// Mitsubishi GX Works2 project: FB_practice   PLC: Q02/Q02H

PROGRAM MAIN
VAR
  DOUBLE_SOL_1 : DOUBLE_SOL;
  DOUBLE_SOL_2 : DOUBLE_SOL;
END_VAR
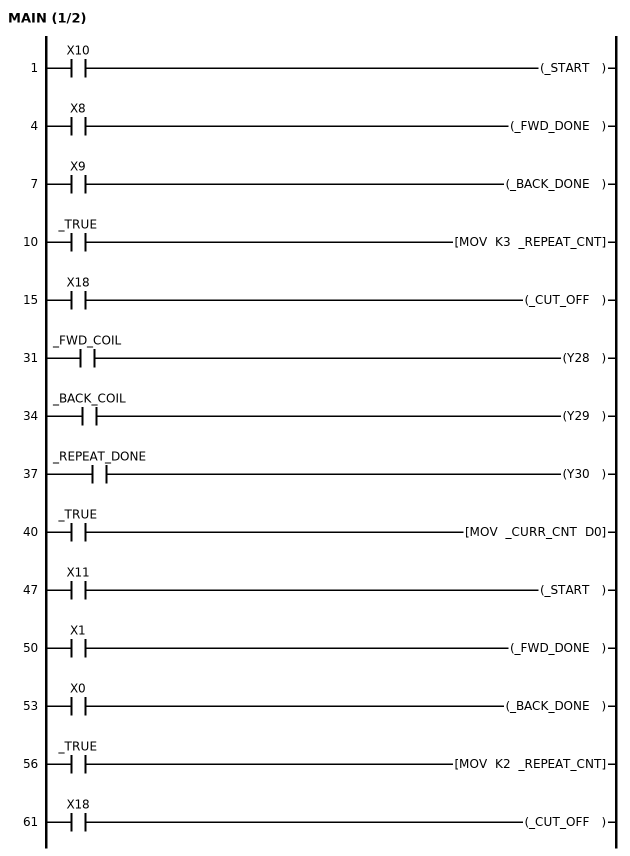
; FB BLK START DOUBLE_SOL(DOUBLE_SOL_1)
1     LD      X10
      OUT     _START
4     LD      X8
      OUT     _FWD_DONE
7     LD      X9
      OUT     _BACK_DONE
10    LD      _TRUE
      MOV     K3 _REPEAT_CNT
15    LD      X18
      OUT     _CUT_OFF
; FB START
; FB_NAME DOUBLE_SOL
; INSTANCE_NAME DOUBLE_SOL_1
; FB IN_B:START
; FB OUT_FWD_COIL:B
; FB IN_B:FWD_DONE
; FB OUT_BACK_COIL:B
; FB IN_B:BACK_DONE
; FB OUT_REPEAT_DONE:B
; FB IN_W:REPEAT_CNT
; FB OUT_CURR_CNT:W
; FB IN_B:CUT_OFF
; FB END
31    LD      _FWD_COIL
      OUT     Y28
34    LD      _BACK_COIL
      OUT     Y29
37    LD      _REPEAT_DONE
      OUT     Y30
40    LD      _TRUE
      MOV     _CURR_CNT D0
; FB BLK END
; FB BLK START DOUBLE_SOL(DOUBLE_SOL_2)
47    LD      X11
      OUT     _START
50    LD      X1
      OUT     _FWD_DONE
53    LD      X0
      OUT     _BACK_DONE
56    LD      _TRUE
      MOV     K2 _REPEAT_CNT
61    LD      X18
      OUT     _CUT_OFF
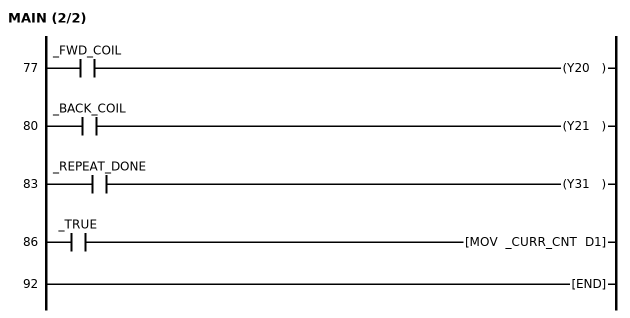
; FB START
; FB_NAME DOUBLE_SOL
; INSTANCE_NAME DOUBLE_SOL_2
; FB IN_B:START
; FB OUT_FWD_COIL:B
; FB IN_B:FWD_DONE
; FB OUT_BACK_COIL:B
; FB IN_B:BACK_DONE
; FB OUT_REPEAT_DONE:B
; FB IN_W:REPEAT_CNT
; FB OUT_CURR_CNT:W
; FB IN_B:CUT_OFF
; FB END
77    LD      _FWD_COIL
      OUT     Y20
80    LD      _BACK_COIL
      OUT     Y21
83    LD      _REPEAT_DONE
      OUT     Y31
86    LD      _TRUE
      MOV     _CURR_CNT D1
; FB BLK END
92    END
END_PROGRAM

FUNCTION_BLOCK DOUBLE_SOL
VAR_INPUT
  START : BOOL;
  FWD_DONE : BOOL;
  BACK_DONE : BOOL;
END_VAR
VAR_OUTPUT
  FWD_COIL : BOOL;
  BACK_COIL : BOOL;
END_VAR
VAR_INPUT
  REPEAT_CNT : INT;
END_VAR
VAR_OUTPUT
  REPEAT_DONE : BOOL;
  CURR_CNT : INT;
END_VAR
VAR_INPUT
  CUT_OFF : BOOL;
END_VAR
VAR
  P_STEP : INT;
END_VAR
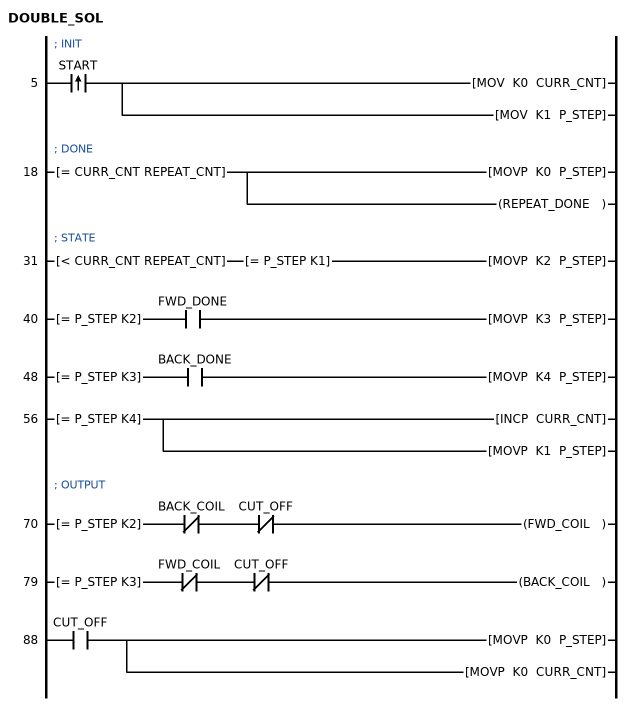
; INIT
5     LDP     START
      MOV     K0 CURR_CNT
      MOV     K1 P_STEP
; DONE
18    LD=     CURR_CNT REPEAT_CNT
      MOVP    K0 P_STEP
      OUT     REPEAT_DONE
; STATE
31    LD<     CURR_CNT REPEAT_CNT
      AND=    P_STEP K1
      MOVP    K2 P_STEP
40    LD=     P_STEP K2
      AND     FWD_DONE
      MOVP    K3 P_STEP
48    LD=     P_STEP K3
      AND     BACK_DONE
      MOVP    K4 P_STEP
56    LD=     P_STEP K4
      INCP    CURR_CNT
      MOVP    K1 P_STEP
; OUTPUT
70    LD=     P_STEP K2
      ANI     BACK_COIL
      ANI     CUT_OFF
      OUT     FWD_COIL
79    LD=     P_STEP K3
      ANI     FWD_COIL
      ANI     CUT_OFF
      OUT     BACK_COIL
88    LD      CUT_OFF
      MOVP    K0 P_STEP
      MOVP    K0 CURR_CNT
END_FUNCTION_BLOCK
